INTERFACE IPistonVertical

METHOD MoveDown : TcoCore.ITcoTaskStatus
END_METHOD

METHOD MoveUp : TcoCore.ITcoTaskStatus
END_METHOD

END_INTERFACE

(* stored: Version 1.1.0.1
   Itf IPistonVertical: Id {d4b15bba-c139-06a8-1cc3-b9c8ec9a5889}
   Folder Vertical: Id {ab932949-6bd4-0eae-030b-f8bd34419e8f}
   Method MoveDown: Id {04784a04-7cc9-012a-26da-ea32fcebfff7}
   Method MoveUp: Id {eeb32c67-58d2-0fef-20ec-7d9b3ff03921} *)
